{attribute 'GeneratedUsingTerminal: EL5151-0000-0020'}
{attribute addProperty BoxType "EL5151-0000-0020"}
{attribute addProperty Id "ENC_InputsAT %I*ENC_Inputs_B353648514ENC_Inputs_1AT %I*ENC_Inputs_24B63C534ENC_OutputsAT %Q*ENC_Outputs_21E2D14D6WcStateAT %I*WcState_9091E0EB2InfoDataAT %I*InfoData_32EB74EA10"}
{attribute addProperty CRC "2421972952"}
{attribute addProperty Size "36"}
TYPE EL5151_905C5FD8 EXTENDS EtcSlaveTerminalBase_947E5A46 :
STRUCT
	{attribute addProperty Name "ENC_Inputs"}
	ENC_Inputs : ENC_Inputs_B3536485;
	{attribute addProperty Name "ENC_Inputs_1"}
	ENC_Inputs_1 : ENC_Inputs_24B63C53;
	{attribute addProperty Name "ENC_Outputs"}
	ENC_Outputs : ENC_Outputs_21E2D14D;
	{attribute addProperty Name "WcState"}
	WcState : WcState_9091E0EB;
	{attribute addProperty Name "InfoData"}
	InfoData : InfoData_32EB74EA;
END_STRUCT
END_TYPE

(* stored: Version 1.2.0.0, ProductVersion 3.1.4024.9
   DUT EL5151_905C5FD8: Id {e4ab8a68-35bd-4fba-8584-ef56a2320dcb} *)
